ABB RobotStudio station: EGM_TCPControl_RW6.16.rspag

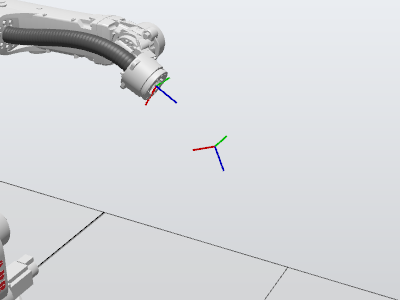
--- station ---
Station EGM_TCPControl_RW6.16 (saved by RobotStudio 25.3.11371.0)
Controller IRB1660ID_4_155
  mechanical unit ROB_1: IRB1660ID_4_155__03, 6 joints, base frame (0, 0, 0) mm
Layout (positions relative to the parent item):
  - IRB1660ID_4_155__03 [mechanism, from %ABB.RobotStudio.Models.IRB1660ID%\IRB1660ID_4_155__03.rslib] at (0, 0, 0) mm; joint values [0, 0, 0, 0, 0.5236, 0] (rad or m)
Targets, tools, work objects and paths stored in the station and not in the controller backup, written as RAPID:
! task T_ROB1
MODULE CalibData
  PERS tooldata MyTool:=[TRUE,[[31.792631019,0,229.638935148],[0.945518576,0,0.325568154,0]],[1,[0,0,1],[1,0,0,0],0,0,0]];
ENDMODULE


--- Controller Data/IRB1660ID_4_155/RAPID/TASK1/PROGMOD/Module1.mod ---
MODULE Module1
    VAR egmident egm_id_tcp;
    LOCAL CONST jointtarget home_pos:=[[0,0,0,0,30,0],[9E9,9E9,9E9,9E9,9E9,9E9]];
    PERS wobjdata egm_wobj:=[FALSE,TRUE,"",[[0,0,0],[1,0,0,0]],[[0,0,0],[1,0,0,0]]];
    PERS tooldata current_tool:=[TRUE,[[0,0,0],[1,0,0,0]],[0.001,[0,0,0.001],[1,0,0,0],0,0,0]];

    ! ??????? ?????????
    LOCAL CONST egm_minmax pose_limits:=[-0.5,0.5];

    LOCAL CONST pose egm_correction_frame:=[[0,0,0],[1,0,0,0]];
    LOCAL CONST pose egm_sensor_frame:=[[0,0,0],[1,0,0,0]];

    PROC main()
        MoveAbsJ home_pos,v200,fine,current_tool;
        InitJointEGM;
        WHILE TRUE DO
            TPWrite "?????? EGM...";
            EGMRunPose egm_id_tcp,
                        EGM_STOP_RAMP_DOWN,
                        \X \Y \Z \Rx \Ry \Rz
                        \CondTime:=1000
                        \RampInTime:=0.05
                        \RampOutTime:=0.5
                        \PosCorrGain:=1.0;
            WaitTime 0.01;
        ENDWHILE
    ENDPROC

    PROC InitJointEGM()
        EGMReset egm_id_tcp;
        EGMGetId egm_id_tcp;

        EGMSetupUC ROB_1,egm_id_tcp,"default","UCdevice1",\Pose\CommTimeout:=5.0;

        EGMActPose egm_id_tcp,
                       \WObj:=egm_wobj,
                       egm_correction_frame,
                       EGM_FRAME_BASE,
                       egm_sensor_frame,
                       EGM_FRAME_BASE
                       \X:=pose_limits
                       \Y:=pose_limits
                       \Z:=pose_limits
                       \Rx:=pose_limits
                       \Ry:=pose_limits
                       \Rz:=pose_limits
                       \LpFilter:=5
                       \SampleRate:=16
                       \MaxPosDeviation:=1000
                       \MaxSpeedDeviation:=30;

    ENDPROC

    PROC StopAll()
        EGMReset egm_id_tcp;
    ENDPROC
ENDMODULE
